{attribute 'linkalways'} 
{attribute 'no_explicit_call' := 'This FB is a CLASS and must be accessed using methods or properties'}
{attribute 'enable_dynamic_creation'}
FUNCTION_BLOCK FINAL TRUNC_LREAL EXTENDS Node
VAR
	in : _LREAL(0.0);
	out : _LREAL(0.0);
END_VAR

METHOD PUBLIC Clone : I_Node
VAR
	pNode : POINTER TO TRUNC_LREAL;
END_VAR
pNode := __NEW(TRUNC_LREAL);
Clone := pNode^;
END_METHOD

METHOD FB_init : BOOL
VAR_INPUT
	bInitRetains : BOOL; // if TRUE, the retain variables are initialized (warm start / cold start)
	bInCopyCode : BOOL;  // if TRUE, the instance afterwards gets moved into the copy code (online change)
END_VAR
AddInput('in',THIS^.in);
AddOutput('out', THIS^.out);
END_METHOD

METHOD PROTECTED OnExecute
VAR
END_VAR
out.Value := LTRUNC(in.Value);
END_METHOD

END_FUNCTION_BLOCK

(* stored: Version 1.1.0.1, ProductVersion 3.1.4024.15
   POU TRUNC_LREAL: Id {49cda9e5-121c-48bf-a5f9-e79b02524187}, SpecialFunc None
   Folder Constructor: Id {6608a611-f556-46fb-b3b6-878060a3d432}
   Method Clone: Id {fc9bab22-963f-4032-81d2-8f65f0026c39}
   Method FB_init: Id {a644416e-2a11-4ae5-a0eb-2fb0e1a10201}
   Method OnExecute: Id {2cc7d3fb-dbcb-44dc-ba76-913b0a8a0406} *)
